{attribute 'GeneratedUsingTerminal: EL2911-0000-0016'}
{attribute addProperty BoxType "EL2911-0000-0016"}
{attribute addProperty Id "OutputsOutputs_A2CAA4461"}
{attribute addProperty CRC "512562743"}
{attribute addProperty Size "1"}
TYPE Module_2_FSOUT_1E8D1637 :
STRUCT
	{attribute addProperty Name "Outputs"}
	Outputs  : Outputs_A2CAA446;
END_STRUCT
END_TYPE

(* stored: Version 1.2.0.0, ProductVersion 3.1.4024.9
   DUT Module_2_FSOUT_1E8D1637: Id {84cca70a-9391-44f5-bbdc-f5c2a1a87ba5} *)
